// TIA Portal V17 export
// export: Created 2025-06-26T06:49:31.1420635Z, ExportSetting WithDefaults, DisplayName Totally Integrated Automation Portal, DisplayVersion V17 Update 8, DisplayName TIA Portal Openness, DisplayVersion V17 Update 8, DisplayName TIA Portal Version Control Interface, DisplayVersion V17, DisplayName STEP 7 Professional, DisplayVersion V17 Update 8, DisplayName STEP 7 Safety, DisplayVersion V17 Update 6, DisplayName WinCC Advanced, DisplayVersion V17 Update 8
TYPE "stSuperheatControl"
// stored: IsFailsafeCompliant false
   STRUCT
      bEnable : Bool;   // 1 = enabled from HMI 0 = disabled from HMI
      bFault : Bool;   // 1 = fault 0 = ok
      nMode : USInt;   // 0 = off, 1 = auto, 2 = manual
      Regulator : "stPID_Regulator_neu";
      fineTuningRecTarget : Real;   // Parameter (0-1). Smaller value will lead to higher power and reduces expander inlet temperatures (superheat), but makes it more instable. The factor in front will increase the (relative) impact
      ExponentialPinchFactor : Real;
      AdditionalSuperheat : Real;
      "FORCE!_FixedPinch" : Bool;
      "FORCE!_FixedPinch_Value" : Real;
   END_STRUCT;
   // Regulator.Kp := 1.0;
   // Regulator.Tn := 1.0;
   // Regulator.Tv := 1.0;
END_TYPE
